ABB RobotStudio station: ABB_conveyor.rspag

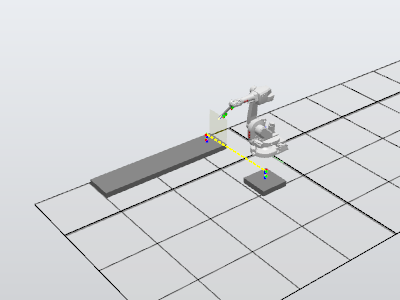
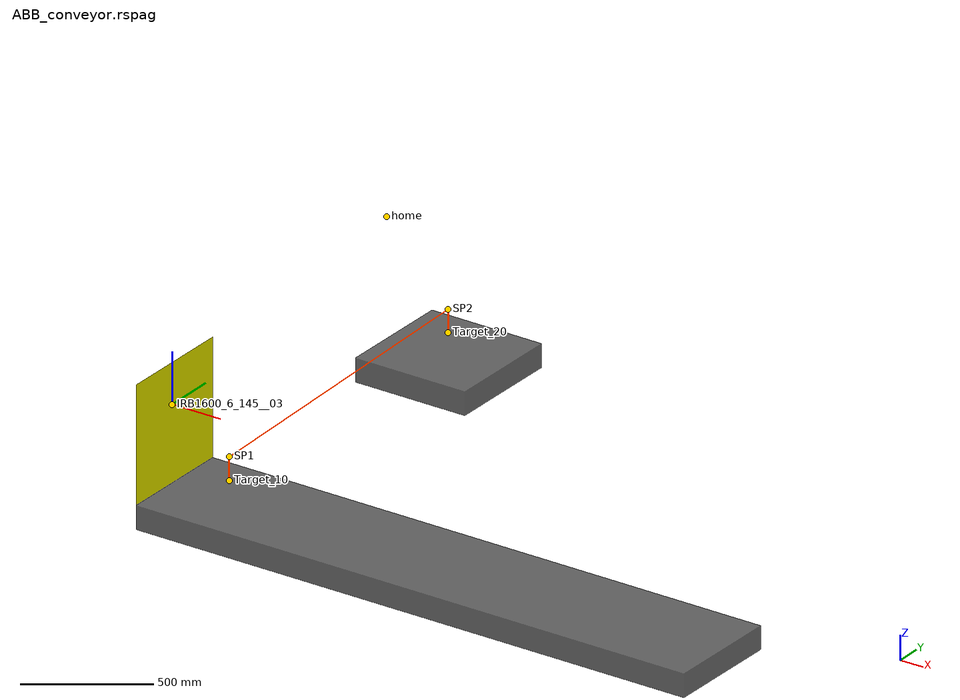
[picture v1: parts stored in the station drawn from their meshes, with robot base, taught points and paths (robot models come from the ABB library and are not in the file)]
--- station ---
Station lab4a_Igor_1 (saved by RobotStudio 24.3.10958.1)
Controller IRB1600_6_145_2
  mechanical unit ROB_1: IRB1600_6_145__03, 6 joints, base frame (0, 0, 0) mm
Layout (positions relative to the parent item):
  - IRB1600_6_145__03 [mechanism, from %ABB.RobotStudio.Models.IRB1600%\IRB1600_6_145_G_03.rslib] at (0, 0, 0) mm; joint values [0, 0, 0, 0, 0.5236, 0] (rad or m)
  - conveyor [part] at (200, 0, 100) mm, size 2500 x 500 x 100 mm
  - bufor [part], size 500 x 500 x 100 mm
  - literka_F [part] at (785, -500, 100) mm, rotated rx 0 ry 0 rz 180 deg, size 288 x 360 x 72 mm
  - PlaneSensor [smart component, from Components\PlaneSensor.rslib]
      properties: Origin=[0.5 -0.45 0.101]; Axis1=[0 0 0.5]; Axis2=[0 -0.5 0]; Tag=(none); SensedPart=(none)
    - _sensorPart_ [part], size 0 x 500 x 500 mm
  - Source [smart component, from Components\Source.rslib]
      properties: Source=literka_F; Copy=(none); Parent=(none); Position=[3 -0.5 0.1]; Orientation=[0 0 3.14159265358979]; Transient=false; PhysicsBehavior=0
  - LinearMover [smart component, from Components\LinearMover.rslib]
      properties: Object=(none); Direction=[-2.5 0 0]; Speed=0.5; Reference=Global; ReferenceObject=(none)
  - Sink [smart component, from Components\Sink.rslib]
      properties: Object=(none)
  - Positioner [smart component, from Components\Positioner.rslib]
      properties: Object=(none); Position=[3 -0.5 0.1]; Orientation=[0 0 3.14159265358979]; Reference=Global; ReferenceObject=(none)
  - SC_VaccumGripper [smart component, from lab3\SC_VaccumGripper.rslib] at (806.29, 0, 1154) mm, rotated rx -180 ry 60 rz -180 deg
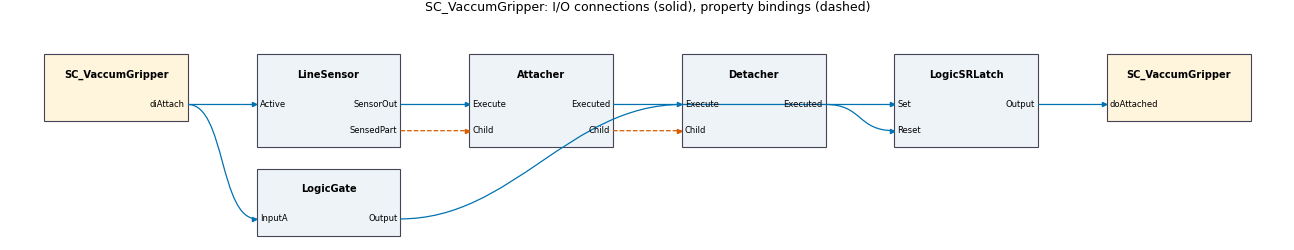
      connections:
        SC_VaccumGripper.diAttach -> LineSensor.Active
        LineSensor.SensorOut -> Attacher.Execute
        Attacher.Executed -> LogicSRLatch.Set
        SC_VaccumGripper.diAttach -> LogicGate.InputA
        LogicGate.Output -> Detacher.Execute
        Detacher.Executed -> LogicSRLatch.Reset
        LogicSRLatch.Output -> SC_VaccumGripper.doAttached
        LineSensor.SensedPart => Attacher.Child
        Attacher.Child => Detacher.Child
    - VaccumGripper [mechanism, from lab3\SC_VaccumGripper.rslib] at (0, 0, 0) mm
    - Attacher [smart component, from Components\Attacher.rslib]
        properties: Parent=VaccumGripper; Flange=0; Child=(none); Mount=false; Offset=[0 0 0]; Orientation=[0 0 0]
    - LineSensor [smart component, from Components\LineSensor.rslib] at (0, 0, 1) mm
        properties: Start=[6.60289067866415E-09 -2.13450085384537E-09 0.200000040663625]; End=[7.4394161941882E-09 -2.24857205077811E-09 0.300000040663625]; Length=0.1; Radius=0.001; Tag=(none); SensedPart=(none); SensedPoint=[0.7 0.8 0.172]
      - _sensorPart_ [part, from lab3\SC_VaccumGripper.rslib]
    - LogicGate [smart component, from Components\LogicGate.rslib]
        properties: Operator=NOT; Delay=0
    - Detacher [smart component, from Components\Detacher.rslib]
        properties: Child=(none); KeepPosition=true
    - LogicSRLatch [smart component, from Components\LogicSRLatch.rslib]
Attachment: VaccumGripper is attached to SC_VaccumGripper
Attachment: SC_VaccumGripper is attached to IRB1600_6_145__03 / Link6
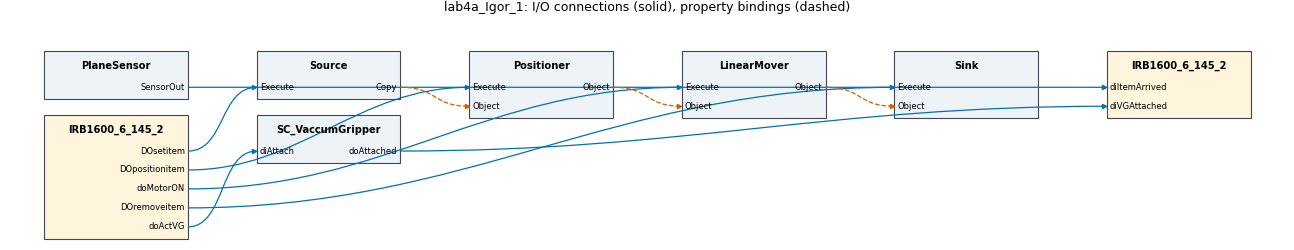
Station logic (signal -> signal, property => property):
  PlaneSensor.SensorOut -> IRB1600_6_145_2.diItemArrived
  IRB1600_6_145_2.DOsetitem -> Source.Execute
  IRB1600_6_145_2.DOpositionitem -> Positioner.Execute
  IRB1600_6_145_2.doMotorON -> LinearMover.Execute
  IRB1600_6_145_2.DOremoveitem -> Sink.Execute
  IRB1600_6_145_2.doActVG -> SC_VaccumGripper.diAttach
  SC_VaccumGripper.doAttached -> IRB1600_6_145_2.diVGAttached
  Source.Copy => Positioner.Object
  Positioner.Object => LinearMover.Object
  LinearMover.Object => Sink.Object

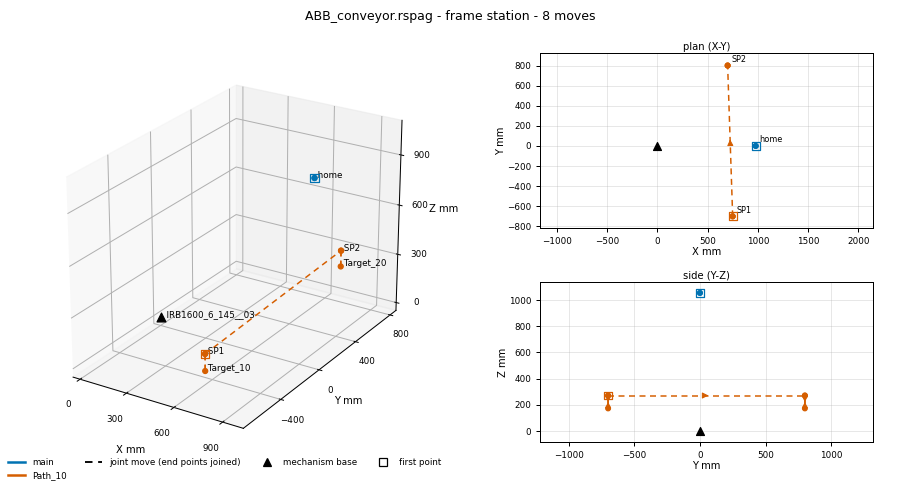
[picture p0: tool path of ABB_conveyor.rspag in frame station, 8 of 8 moves have a stored position in this frame; points joined in program order, loops and branches not executed]
--- Backups/IRB1600_6_145_2/RAPID/TASK1/PROGMOD/CalibData.mod ---
MODULE CalibData
    PERS tooldata gripper_MH:=[TRUE,[[0,0,150],[1,0,0,0]],[0.375,[0,0,75],[1,0,0,0],0.00078125,0.00078125,0.00015625]];
    PERS tooldata VaccumGripper_TCP:=[TRUE,[[0,0,200],[1,0,0,0]],[0.18,[0,0,100],[1,0,0,0],0.0006135,0.0006135,0.000027]];
ENDMODULE

--- Backups/IRB1600_6_145_2/RAPID/TASK1/PROGMOD/Module1.mod ---
MODULE Module1
        CONST robtarget SP1:=[[750,-700,272],[0,1,0,0],[0,0,0,0],[9E+09,9E+09,9E+09,9E+09,9E+09,9E+09]];
    CONST robtarget Target_10:=[[750,-700,173.5],[0,1,0,0],[0,0,0,0],[9E+09,9E+09,9E+09,9E+09,9E+09,9E+09]];
    CONST robtarget SP2:=[[700,800,272],[0,0,1,0],[0,0,0,0],[9E+09,9E+09,9E+09,9E+09,9E+09,9E+09]];
    CONST robtarget Target_20:=[[700,800,173.5],[0,0,1,0],[0,0,0,0],[9E+09,9E+09,9E+09,9E+09,9E+09,9E+09]];
    CONST robtarget home:=[[979.496732003,0,1054],[0.5,0,0.866025404,0],[0,0,0,0],[9E+09,9E+09,9E+09,9E+09,9E+09,9E+09]];
!***********************************************************
    !
    ! Module:  Module1
    !
    ! Description:
    !   <Insert description here>
    !
    ! Author: Igor Cena
    !
    ! Version: 1.0
    !
    !***********************************************************


    !***********************************************************
    !
    ! Procedure main
    !
    !   This is the entry point of your program
    !
    !***********************************************************
    PROC main()
        MoveJ home,v400,z100,VaccumGripper_TCP\WObj:=wobj0;
        SetDO doActVG,0;
        SetDO doMotorON,0;
        SetDO DOpositionitem,0;
        SetDO DOremoveitem,0;
        SetDO DOsetitem,0;
        SetDO DOsetitem,1;
        SetDO DOsetitem,0;
        SetDO doMotorON,1;
        WaitDI diItemArrived,1;
        SetDO doMotorON, 0;
        Path_10;
        MoveJ home,v400,z100,VaccumGripper_TCP\WObj:=wobj0;
        SetDO DOremoveitem,1;
    ENDPROC
    PROC Path_10()
        MoveJ SP1,v400,z100,VaccumGripper_TCP\WObj:=wobj0;
        MoveJ Target_10,v400,fine,VaccumGripper_TCP\WObj:=wobj0;
        Grasp;
        MoveJ SP1,v400,z100,VaccumGripper_TCP\WObj:=wobj0;
        MoveJ SP2,v400,z100,VaccumGripper_TCP\WObj:=wobj0;
        MoveJ Target_20,v400,fine,VaccumGripper_TCP\WObj:=wobj0;
        Release;
        MoveJ SP2,v400,z100,VaccumGripper_TCP\WObj:=wobj0;
    ENDPROC
PROC Grasp()
 WaitTime 1;
 SetDO doActVG,1;
 WaitTime 1;
 WaitDI diVGAttached,1;
 ENDPROC
 PROC Release()
 WaitTime 1;
 SetDO doActVG,0;
 WaitTime 1;
 WaitDI diVGAttached,0;
 ENDPROC
ENDMODULE

--- Backups/IRB1600_6_145_2/SYSPAR/EIO.cfg ---
EIO:CFG_1.0:6:1::
#
INDUSTRIAL_NETWORK:

      -Name "DeviceNet" -Label "DeviceNet Master/Slave Network" -Address "2"
#
DEVICENET_DEVICE:

      -Name "d652" -VendorName "ABB Robotics" -ProductName "24 VDC I/O Device"\
      -Label "DSQC 652 24 VDC I/O Device" -ProductCode 26 -DeviceType 7\
      -ConnectionType "COS" -OutputSize 2 -InputSize 2
#
DEVICENET_INTERNAL_DEVICE:

      -Name "DN_Internal_Device" -VendorName "ABB Robotics"\
      -ProductName "DeviceNet Internal Slave Device"
#
EIO_SIGNAL:

      -Name "doActVG" -SignalType "DO" -Device "d652"\
      -Label "sets gripper on/off" -DeviceMap "0"

      -Name "doMotorON" -SignalType "DO" -Device "d652"\
      -Label "starts conveyor motion" -DeviceMap "1"

      -Name "diVGAttached" -SignalType "DI" -Device "d652" -Label "item grasped"\
      -DeviceMap "0"

      -Name "diItemArrived" -SignalType "DI" -Device "d652"\
      -Label "item ready for manipulation" -DeviceMap "1"

      -Name "DOpositionitem" -SignalType "DO"\
      -Label "positions item on conveyor"

      -Name "DOremoveitem" -SignalType "DO" -Label "removes item"

      -Name "DOsetitem" -SignalType "DO" -Label "makes copy of item"
